FUNCTION Convert_TOD_TO_DWORD : Hresult
VAR_INPUT
	in : TOD;
	out : REFERENCE TO DWORD;
END_VAR
VAR
	converted : DWORD;
END_VAR

converted := TOD_TO_DWORD(in);

IF (DWORD_TO_TOD(converted) <> in) THEN
	Convert_TOD_TO_DWORD := INCOMPATIBLE;
	RETURN;
END_IF

out := converted;

END_FUNCTION

(* stored: Version 1.1.0.1, ProductVersion 3.1.4024.12
   POU Convert_TOD_TO_DWORD: Id {1cfdce1d-9404-4912-9733-03b577a9cdf5}, SpecialFunc None *)
